PROGRAM MAIN
VAR
	TC_RST				:	TC_Restart;
	ClrMem_Trig			:	R_TRIG;	
	LightsTime			:	TON;
END_VAR

TC_RST(RESTART := GVL_Main.IN.PlcReset, TMOUT := T#5S);		//Reset PLC from HMI

ClrMem_Trig(CLK := (NOT GVL_Main.Estop));
IF ClrMem_Trig.Q THEN									//Make all HMI commands false when Estop
	MEMSET(ADR(GVL_Main.IN), 0, SIZEOF(GVL_Main.IN));
END_IF

IF NOT GVL_Main.Estop THEN
	GVL_Main.OUT.RoutineResetFeedback	:=	0;
	GVL_Main.OUT.InitializeFeedback		:=	0;
	GVL_Main.OUT.NextFeedback			:=	0;
	GVL_Main.OUT.RunFeedback			:=	0;
	GVL_Main.OUT.StationFeedback		:=	0;
	GVL_Main.OUT.ClearErrorFeedback		:=	0;
	GVL_Main.OUT.RoutineResetDone		:=	0;
	GVL_Main.OUT.InitializeDone			:=	0;
	
	IF GVL_Main.DoorClosed THEN
		GVL_Main.MachineLights := FALSE;
		IF LightsTime.Q THEN
			LightsTime(IN := FALSE, PT := T#1000MS);
			IF GVL_Main.EstopLights THEN
			//IF GVL_Main.MachineLights THEN
				GVL_Main.EstopLights := FALSE;
				//GVL_Main.MachineLights := FALSE;
			ELSE
				GVL_Main.EstopLights := TRUE;
				//GVL_Main.MachineLights := TRUE;
			END_IF
		ELSE
			LightsTime(IN := TRUE, PT := T#1000MS);
		END_IF
	ELSE
		GVL_Main.EstopLights := FALSE;
		GVL_Main.MachineLights := TRUE;
	END_IF
	
	//reset routine for all the stations
	STATION_01(ExecuteAll := FALSE);
	STATION_02(ExecuteAll := FALSE);
	STATION_03(ExecuteAll := FALSE);
	STATION_04(ExecuteAll := FALSE);
	STATION_05(ExecuteAll := FALSE);
	STATION_06(ExecuteAll := FALSE);
	STATION_07(ExecuteAll := FALSE);
	STATION_08(ExecuteAll := FALSE);
	STATION_09(ExecuteAll := FALSE);
	
ELSE
	//Estop Lights
	GVL_Main.EstopLights := FALSE;
	//Machine Lights
	//GVL_Main.MachineLights := TRUE;
	//All station programs here
	STATION_01(ExecuteAll := TRUE);
	STATION_02(ExecuteAll := TRUE);
	STATION_03(ExecuteAll := TRUE);
	STATION_04(ExecuteAll := TRUE);
	STATION_05(ExecuteAll := TRUE);
	STATION_06(ExecuteAll := TRUE);
	STATION_07(ExecuteAll := TRUE);
	STATION_08(ExecuteAll := TRUE);
	STATION_09(ExecuteAll := TRUE);
	
	(*Warning Lights*)
	IF GVL_Main.OUT.RunError > 0 THEN
		IF GVL_Main.DoorClosed THEN
			IF LightsTime.Q THEN
				LightsTime(IN := FALSE, PT := T#1000MS);
				IF GVL_Main.MachineLights THEN
					GVL_Main.MachineLights := FALSE;
				ELSE
					GVL_Main.MachineLights := TRUE;
				END_IF
			ELSE
				LightsTime(IN := TRUE, PT := T#1000MS);
			END_IF
		ELSE
			GVL_Main.MachineLights := TRUE;
		END_IF
	ELSE
		GVL_Main.MachineLights := TRUE;
	END_IF
	
END_IF

END_PROGRAM

(* stored: Version 1.1.0.1, ProductVersion 3.1.4020.12
   POU MAIN: Id {f75c814b-849c-450c-86c8-4df41ee853fe}, SpecialFunc None *)
